Fanuc KAREL source: BYTES_LEFT.kl

PROGRAM T
%NOLOCKGROUP
VAR
 v0 : FILE
 res : INTEGER
BEGIN
 res = BYTES_LEFT(v0)
END T
